PROGRAM MAIN
VAR

	lamp: BOOL;

	
END_VAR



IF GVL.light = TRUE THEN
	lamp := TRUE;
ELSE
	lamp := FALSE;
END_IF

END_PROGRAM

(* stored: Version 1.1.0.1, ProductVersion 3.1.4024.12
   POU MAIN: Id {f7fde937-a145-4461-be69-639376c0a1a8}, SpecialFunc None *)
